ADAPTER AdpChan (* Adapter Interface *)
  (* Standard: 61499-1 *)
  (* Version 0.0, 12/6/2023, vaatmar1, nxtControl GmBH *)
  PACKAGE Main;
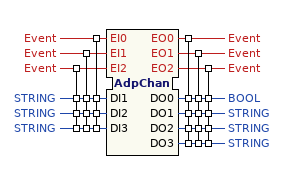
  EVENT_INPUT
    EI0 WITH DI1, DI2, DI3;
    EI1 WITH DI1, DI2, DI3;
    EI2 WITH DI1, DI2, DI3;
  END_EVENT
  EVENT_OUTPUT
    EO0 WITH DO0, DO1, DO2, DO3;
    EO1 WITH DO0, DO1, DO2, DO3;
    EO2 WITH DO0, DO1, DO2, DO3;
  END_EVENT
  VAR_INPUT
    DI1 : STRING;
    DI2 : STRING;
    DI3 : STRING;
  END_VAR
  VAR_OUTPUT
    DO0 : BOOL;
    DO1 : STRING;
    DO2 : STRING;
    DO3 : STRING;
  END_VAR
  SERVICE SOCKET/PLUG
    SEQUENCE request_confirm
      SOCKET.REQ(REQD) -> PLUG.REQ(REQD);
      PLUG.CNF(CNFD) -> SOCKET.CNF(CNFD);
    END_SEQUENCE
    SEQUENCE indication_response
      PLUG.IND(INDD) -> SOCKET.IND(INDD);
      SOCKET.RSP(RSPD) -> PLUG.RSP(RSPD);
    END_SEQUENCE
  END_SERVICE
END_ADAPTER
